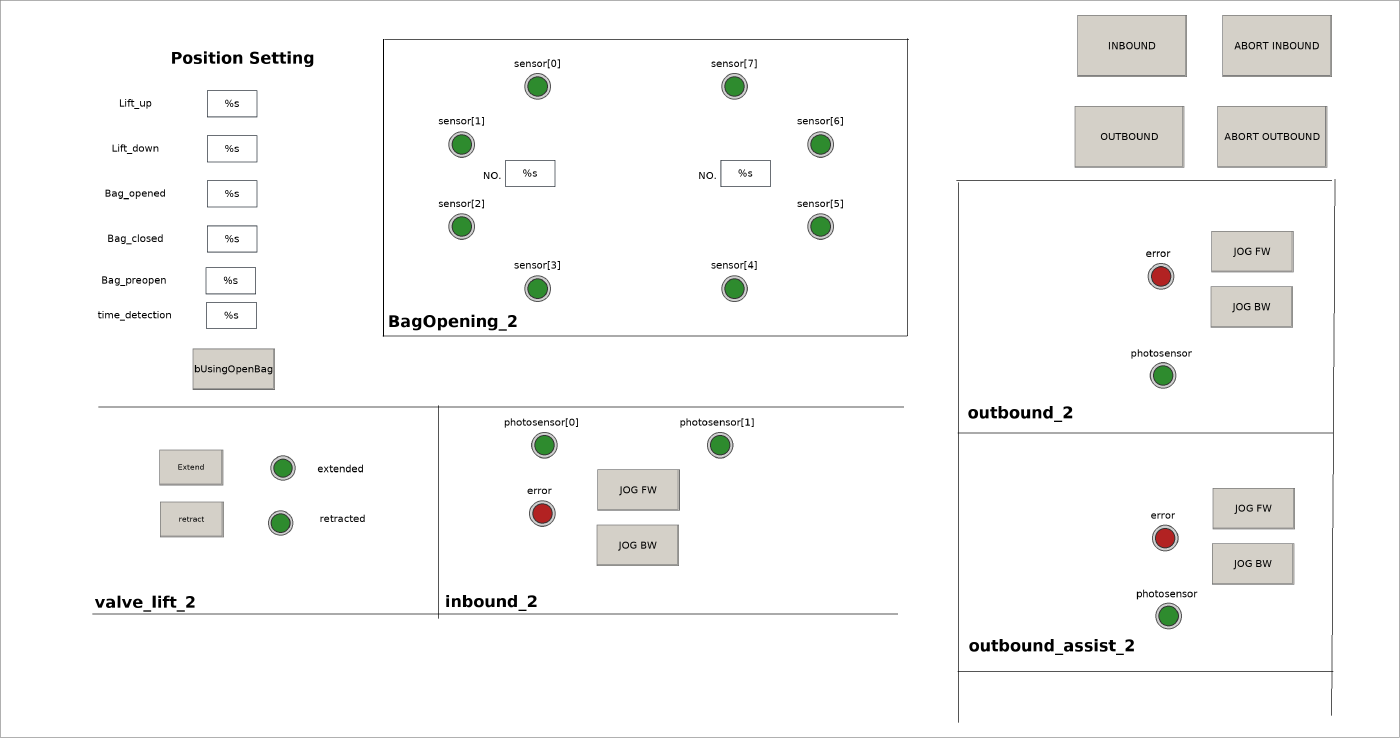
VISUALIZATION v_io_working2  // 2048x1080
    Label (91,855 244x53), "valve_lift_2"
    Button (233,658 93x52), "Extend", colour toggle: GVL.fb_working1.valve_lift.extend
        OnMouseDown: execute { GVL.fb_working2.valve_lift.extend := TRUE; GVL.fb_working2.valve_lift.retract := FALSE; }
    Button (234,734 93x52), "retract", colour toggle: GVL.fb_working1.valve_lift.retract
        OnMouseDown: execute { GVL.fb_working2.valve_lift.extend 	:= FALSE; GVL.fb_working2.valve_lift.retract 	:= TRUE; }
    Lamp1 (387,664 54x42), variable: GVL.fb_working2.valve_lift.extended, style: Lamp-Lamp1-Green
    Lamp1 (387,744 47x43), variable: GVL.fb_working2.valve_lift.retracted, style: Lamp-Lamp1-Green
    Label (432,673 132x26), "extended"
    Label (435,746 132x26), "retracted"
    Lamp1 (771,729 45x45), variable: GVL.fb_working2.roller_inbound.roller.err.Q, style: Lamp-Lamp1-Red
    Label (689,705 200x26), "error"
    Line (144,595) (1322,595)
    Button (874,687 120x60), "JOG FW", colour toggle: GVL.fb_working1.roller_inbound.roller.forward
        OnMouseDown: execute { GVL.fb_working2.roller_inbound.roller.forward	:= TRUE; }
        OnMouseUp: execute { GVL.fb_working2.roller_inbound.roller.forward	:= FALSE; }
    Button (873,768 120x60), "JOG BW", colour toggle: GVL.fb_working1.roller_inbound.roller.backward
        OnMouseDown: execute { GVL.fb_working2.roller_inbound.roller.backward	:= TRUE; }
        OnMouseUp: execute { GVL.fb_working2.roller_inbound.roller.backward	:= FALSE; }
    Lamp1 (774,629 45x45), variable: GVL.fb_working2.roller_inbound.photo_sensor[0].Q, style: Lamp-Lamp1-Green
    Label (692,605 200x26), "photosensor[0]"
    Lamp1 (1031,629 45x45), variable: GVL.fb_working2.roller_inbound.photo_sensor[1].Q, style: Lamp-Lamp1-Green
    Label (949,605 200x26), "photosensor[1]"
    Label (607,855 224x51), "inbound_2"
    Lamp1 (1676,382 45x45), variable: GVL.fb_working2.roller_outbound.roller.err.Q, style: Lamp-Lamp1-Red
    Label (1594,358 200x26), "error"
    Line (1399,264) (1948,264)
    Button (1772,338 120x60), "JOG FW", colour toggle: GVL.fb_working1.roller_outbound.roller.forward
        OnMouseDown: execute { GVL.fb_working2.roller_outbound.roller.forward	:= TRUE; }
        OnMouseUp: execute { GVL.fb_working2.roller_outbound.roller.forward	:= FALSE; }
    Button (1771,419 120x60), "JOG BW", colour toggle: GVL.fb_working1.roller_outbound.roller.backward
        OnMouseDown: execute { GVL.fb_working2.roller_outbound.roller.backward	:= TRUE; }
        OnMouseUp: execute { GVL.fb_working2.roller_outbound.roller.backward	:= FALSE; }
    Label (1375,587 236x34), "outbound_2"
    Lamp1 (1682,765 45x45), variable: GVL.fb_working2.roller_outbound_assist.roller.err.Q, style: Lamp-Lamp1-Red
    Label (1601,741 200x26), "error"
    Line (1401,633) (1950,633)
    Button (1774,714 120x60), "JOG FW", colour toggle: GVL.fb_working1.roller_outbound_assist.roller.forward
        OnMouseDown: execute { GVL.fb_working2.roller_outbound_assist.roller.forward	:= TRUE; }
        OnMouseUp: execute { GVL.fb_working2.roller_outbound_assist.roller.forward	:= FALSE; }
    Button (1773,795 120x60), "JOG BW", colour toggle: GVL.fb_working1.roller_outbound_assist.roller.backward
        OnMouseDown: execute { GVL.fb_working1.roller_outbound_assist.roller.backward	:= TRUE; }
        OnMouseUp: execute { GVL.fb_working1.roller_outbound_assist.roller.backward	:= FALSE; }
    Line (1401,982) (1950,982)
    Label (1352,940 374x68), "outbound_assist_2"
    Line (641,905) (641,593)
    Line (1948,1047) (1953,262)
    Line (1402,1057) (1402,267)
    Line (135,898) (1313,898)
    Lamp1 (764,400 45x45), variable: GVL.fb_working2.BagOpening_Detection[3], style: Lamp-Lamp1-Green
    Label (686,375 200x26), "sensor[3]"
    Lamp1 (1052,400 45x45), variable: GVL.fb_working2.BagOpening_Detection[4], style: Lamp-Lamp1-Green
    Label (974,375 200x26), "sensor[4]"
    Lamp1 (1178,309 45x45), variable: GVL.fb_working2.BagOpening_Detection[5], style: Lamp-Lamp1-Green
    Label (1100,285 200x26), "sensor[5]"
    Lamp1 (1178,189 45x45), variable: GVL.fb_working2.BagOpening_Detection[6], style: Lamp-Lamp1-Green
    Label (1100,164 200x26), "sensor[6]"
    Lamp1 (1052,104 45x45), variable: GVL.fb_working2.BagOpening_Detection[7], style: Lamp-Lamp1-Green
    Label (974,80 200x26), "sensor[7]"
    Lamp1 (764,104 45x45), variable: GVL.fb_working2.BagOpening_Detection[0], style: Lamp-Lamp1-Green
    Label (686,80 200x26), "sensor[0]"
    Lamp1 (653,189 45x45), variable: GVL.fb_working2.BagOpening_Detection[1], style: Lamp-Lamp1-Green
    Label (575,164 200x26), "sensor[1]"
    Lamp1 (653,309 45x45), variable: GVL.fb_working2.BagOpening_Detection[2], style: Lamp-Lamp1-Green
    Label (575,285 200x26), "sensor[2]"
    Line (562,57) (1329,57)
    Line (561,492) (561,57)
    Line (560,491) (1327,491)
    Line (1328,491) (1328,56)
    Rectangle (303,132 73x39), "%s", text variable: GVL.fb_working2.rPos_lift_up
        OnMouseClick: write the text variable via Default, min GVL.fb_working1.rMin_lift, max GVL.fb_working1.rMax_lift
    Rectangle (303,198 73x39), "%s", text variable: GVL.fb_working2.rPos_lift_down
        OnMouseClick: write the text variable via Default, min GVL.fb_working1.rMin_lift, max GVL.fb_working1.rMax_lift
    Rectangle (303,264 73x39), "%s", text variable: GVL.fb_working2.rPos_bag_opened
        OnMouseClick: write the text variable via Default, min GVL.fb_working1.rMin_bag, max GVL.fb_working1.rMax_bag
    Rectangle (303,330 73x39), "%s", text variable: GVL.fb_working2.rPos_bag_closed
        OnMouseClick: write the text variable via Default, min GVL.fb_working1.rMin_bag, max GVL.fb_working1.rMax_bag
    Label (98,138 200x26), "Lift_up"
    Label (98,204 200x26), "Lift_down"
    Label (98,270 200x26), "Bag_opened"
    Label (98,336 200x26), "Bag_closed"
    Label (180,72 350x26), "Position Setting"
    Rectangle (739,234 73x39), "%s", text variable: GVL.fb_working2.iSensor_detection_setting[0]
        OnMouseClick: write the text variable via Default, min 3, max 4
    Label (670,244 100x26), "NO."
    Rectangle (1054,234 73x39), "%s", text variable: GVL.fb_working2.iSensor_detection_setting[1]
        OnMouseClick: write the text variable via Default, min 3, max 4
    Label (985,244 100x26), "NO."
    Label (447,416 432x109), "BagOpening_2"
    Lamp1 (1679,527 45x45), variable: GVL.fb_working2.photo_sensor_tote_detection.Q, style: Lamp-Lamp1-Green
    Label (1599,504 200x26), "photosensor"
    Lamp1 (1687,879 45x45), variable: GVL.fb_working2.roller_outbound.photo_sensor.Q, style: Lamp-Lamp1-Green
    Label (1607,856 200x26), "photosensor"
    Rectangle (301,391 73x39), "%s", text variable: GVL.fb_working2.rPos_bag_preopen
        OnMouseClick: write the text variable via Default, min GVL.fb_working2.rMin_bag, max 15
    Label (96,397 200x26), "Bag_preopen"
    Rectangle (302,442 73x39), "%s", text variable: GVL.fb_working2.iDelay_sensor_detection
        OnMouseClick: write the text variable via Default, min 100, max 500
    Label (97,448 200x26), "time_detection"
    Button (1576,22 160x90), "INBOUND", colour toggle: MAIN.tote_2.bInbound
        OnMouseUp: execute { MAIN.tote_2.bInbound	:= TRUE; }
    Button (1572,155 160x90), "OUTBOUND", colour toggle: MAIN.tote_2.bOutbound
        OnMouseUp: execute { MAIN.tote_2.bOutbound	:= TRUE; }
    Button (1788,22 160x90), "ABORT INBOUND", colour toggle: MAIN.tote_2.bAbortInbound
        OnMouseUp: execute { MAIN.tote_2.bAbortInbound	:= TRUE; }
    Button (1781,155 160x90), "ABORT OUTBOUND", colour toggle: MAIN.tote_2.bAbortOutbound
        OnMouseUp: execute { MAIN.tote_2.bAbortOutbound	:= TRUE; }
    Button (282,510 120x60), "bUsingOpenBag", colour toggle: GVL.fb_working2.bUsingOpenBag
        toggle GVL.fb_working2.bUsingOpenBag
END_VISUALIZATION

(* stored: Version 1.1.0.1, ProductVersion 3.1.4024.12
   Visu v_io_working2: Id {e0079962-c3ec-4c31-b3bc-1dc0334b31c3} *)
